Staubli VAL3: MX1_NETWORK.dtx

mdesc mNomSpeed
sio sSocket1 = {link=Socket\sock1}
